{attribute 'enable_dynamic_creation'}
FUNCTION_BLOCK CommandNull IMPLEMENTS I_Command
VAR_INPUT
END_VAR
VAR_OUTPUT
END_VAR

METHOD Destroy
VAR_INPUT
END_VAR
END_METHOD

METHOD PUBLIC Execute : BOOL
VAR_INPUT
END_VAR
END_METHOD

PROPERTY PUBLIC hasTimedOut : BOOL
GET
hasTimedOut := false;
END_GET
END_PROPERTY

PROPERTY PUBLIC isBusy : BOOL
GET
isBusy := false;
END_GET
END_PROPERTY

PROPERTY isComplete : BOOL
GET
isComplete := true;
END_GET
END_PROPERTY

END_FUNCTION_BLOCK

(* stored: Version 1.1.0.1, ProductVersion 3.1.4024.9
   POU CommandNull: Id {b4285bea-1d50-47de-b401-5784283591d5}, SpecialFunc None
   Method Destroy: Id {6e92e4e7-b63b-42bb-a5c0-163dc03d8235}
   Method Execute: Id {f61e9aab-f248-489d-b401-3b5d77cce9c1}
   Property hasTimedOut: Id {a84dc935-cceb-42e4-a12d-774e04a4b62e}
   Get Get: Id {5ddf4554-bd96-4cd9-8d17-fa33f194dfdf}
   Property isBusy: Id {effb71e0-3c4a-4ac7-8f0a-91656c359ae8}
   Get Get: Id {fb967f08-8b66-4e5a-a6eb-f89b5d5da71a}
   Property isComplete: Id {dc62dada-a87c-48b3-9261-2a693ff063b1}
   Get Get: Id {125bebac-0933-4b8b-8484-ff5a645b64bf} *)
